FUNCTION_BLOCK OPC_Client (* Simple FB with one algorithm *)
  (* Standard: 61499-1 *)
  (* Version 1.0, 2025-07-18, vadim *)
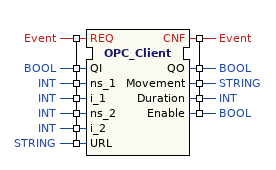
  EVENT_INPUT
    REQ WITH ns_1, i_1, ns_2, i_2, QI, URL; (* Normal Execution Request *)
  END_EVENT
  EVENT_OUTPUT
    CNF WITH Movement, Duration, QO, Enable; (* Execution Confirmation *)
  END_EVENT
  VAR_INPUT
    QI : BOOL;
    ns_1 : INT; (* ns for first var *)
    i_1 : INT; (* i for first var *)
    ns_2 : INT; (* ns for second var *)
    i_2 : INT; (* i for second var *)
    URL : STRING; (* OPC-server URL *)
  END_VAR
  VAR_OUTPUT
    QO : BOOL;
    Movement : STRING; (* Kind of movement *)
    Duration : INT; (* Duration (ms) *)
    Enable : BOOL; (* Enable to start movement *)
  END_VAR
  EC_STATES
    REQ : REQ -> CNF;
  END_STATES
  ALGORITHM REQ IN ST:

  END_ALGORITHM
END_FUNCTION_BLOCK
